// SIMATIC STEP 7 (V5.x) project BatTatTheoNhietDo_PT100
// CPU: CPU 314C-2 DP
// station: Hardware
// station: SIMATIC 300(1)
// station: P_ADR_BUS
// program: S7 Program(1)

SYMBOL_TABLE
"Bat quat mem"	M 0.0	BOOL
"Tat quat mem"	M 0.1	BOOL
"Bat den mem"	M 0.2	BOOL
"Tat den mem"	M 0.3	BOOL
"Auto"	M 0.4	BOOL
"Manual"	M 0.5	BOOL
"Quat_clone_auto"	M 0.6	BOOL
"Den_clone_auto"	M 0.7	BOOL
"Quat_clone_manual"	M 1.0	BOOL
"Den_clone_manula"	M 1.1	BOOL
"model"	M 1.2	BOOL
"Quat"	Q 0.0	BOOL
"Den"	Q 0.1	BOOL
END_SYMBOL_TABLE
